PROGRAM AutoMode
VAR
END_VAR

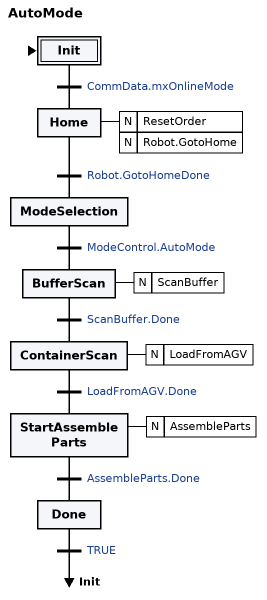
INITIAL_STEP Init:
END_STEP
TRANSITION FROM Init TO Home
    := CommData.mxOnlineMode;
END_TRANSITION
STEP Home:
    ResetOrder(N);
    Robot.GotoHome(N);
END_STEP
TRANSITION FROM Home TO ModeSelection
    := Robot.GotoHomeDone;
END_TRANSITION
STEP ModeSelection:
END_STEP
TRANSITION FROM ModeSelection TO BufferScan
    := ModeControl.AutoMode;
END_TRANSITION
STEP BufferScan:
    ScanBuffer(N);
END_STEP
TRANSITION FROM BufferScan TO ContainerScan
    := ScanBuffer.Done;
END_TRANSITION
STEP ContainerScan:
    LoadFromAGV(N);
END_STEP
TRANSITION FROM ContainerScan TO StartAssembleParts
    := LoadFromAGV.Done;
END_TRANSITION
STEP StartAssembleParts:
    AssembleParts(N);
END_STEP
TRANSITION FROM StartAssembleParts TO Done
    := AssembleParts.Done;
END_TRANSITION
STEP Done:
END_STEP
TRANSITION FROM Done TO Init
    := TRUE;
END_TRANSITION

ACTION ResetOrder:
GVL.qsOrderFornextAssembly := '0';
END_ACTION

ACTION ResetVars:
GVL.BufferProducts.Storage1.Component := '';
GVL.BufferProducts.Storage1.Quatity := 0;
GVL.BufferProducts.Storage2.Component := '';
GVL.BufferProducts.Storage2.Quatity := 0;
GVL.BufferProducts.Storage3.Component := '';
GVL.BufferProducts.Storage3.Quatity := 0;
END_ACTION

END_PROGRAM

(* stored: Version 1.1.0.1, ProductVersion 3.1.4024.12
   POU AutoMode: Id {e4a8051c-91ba-46c4-9c7c-65fd987bbcba}, SpecialFunc None
   Action ResetOrder: Id {263b1f63-e4c6-416c-992d-a77eaac9309e}
   Action ResetVars: Id {1d6e026e-0341-43c4-8f6f-a9d599d4139e} *)
